FUNCTION_BLOCK FB_Discharger_SFC EXTENDS FB_Object_Template_SFC
VAR_INPUT
	B1: BOOL;
	B2: BOOL;
	dcha_1: BOOL;
	dcha_2: BOOL;
	izda_1: BOOL;
	izda_2: BOOL;
	arriba: BOOL;
	abajo: BOOL;
	cogido: BOOL;
END_VAR
VAR_OUTPUT
	avanza_1: BOOL;
	avanza_2: BOOL;
	baja: BOOL;
	coge: BOOL;
END_VAR
VAR
END_VAR

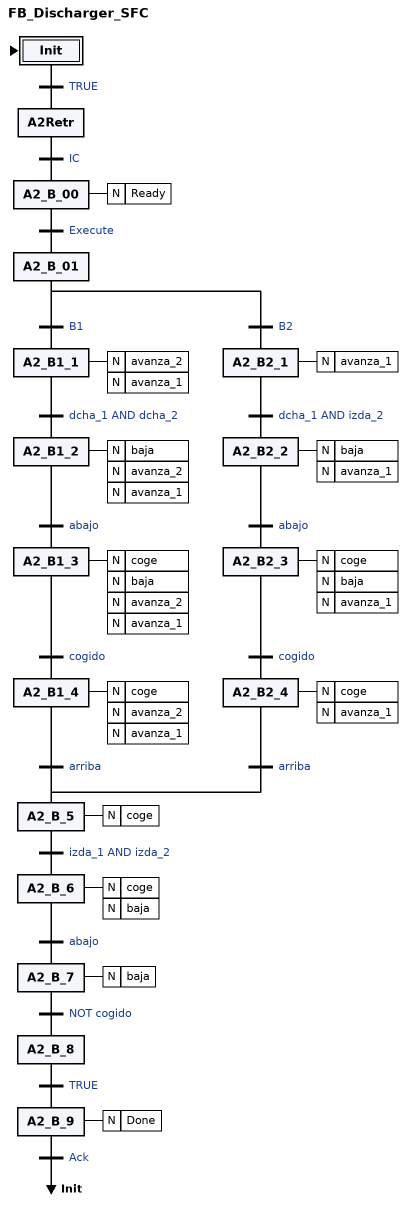
INITIAL_STEP Init:
END_STEP
TRANSITION FROM Init TO A2Retr
    := TRUE;
END_TRANSITION
STEP A2Retr:
END_STEP
TRANSITION FROM A2Retr TO A2_B_00
    := IC;
END_TRANSITION
STEP A2_B_00:
    Ready(N);
END_STEP
TRANSITION FROM A2_B_00 TO A2_B_01
    := Execute;
END_TRANSITION
STEP A2_B_01:
END_STEP
TRANSITION FROM A2_B_01 TO A2_B1_1
    := B1;
END_TRANSITION
STEP A2_B1_1:
    avanza_2(N);
    avanza_1(N);
END_STEP
TRANSITION FROM A2_B1_1 TO A2_B1_2
    := dcha_1 AND dcha_2;
END_TRANSITION
STEP A2_B1_2:
    baja(N);
    avanza_2(N);
    avanza_1(N);
END_STEP
TRANSITION FROM A2_B1_2 TO A2_B1_3
    := abajo;
END_TRANSITION
STEP A2_B1_3:
    coge(N);
    baja(N);
    avanza_2(N);
    avanza_1(N);
END_STEP
TRANSITION FROM A2_B1_3 TO A2_B1_4
    := cogido;
END_TRANSITION
STEP A2_B1_4:
    coge(N);
    avanza_2(N);
    avanza_1(N);
END_STEP
TRANSITION FROM A2_B1_4 TO A2_B_5
    := arriba;
END_TRANSITION
TRANSITION FROM A2_B_01 TO A2_B2_1
    := B2;
END_TRANSITION
STEP A2_B2_1:
    avanza_1(N);
END_STEP
TRANSITION FROM A2_B2_1 TO A2_B2_2
    := dcha_1 AND izda_2;
END_TRANSITION
STEP A2_B2_2:
    baja(N);
    avanza_1(N);
END_STEP
TRANSITION FROM A2_B2_2 TO A2_B2_3
    := abajo;
END_TRANSITION
STEP A2_B2_3:
    coge(N);
    baja(N);
    avanza_1(N);
END_STEP
TRANSITION FROM A2_B2_3 TO A2_B2_4
    := cogido;
END_TRANSITION
STEP A2_B2_4:
    coge(N);
    avanza_1(N);
END_STEP
TRANSITION FROM A2_B2_4 TO A2_B_5
    := arriba;
END_TRANSITION
STEP A2_B_5:
    coge(N);
END_STEP
TRANSITION FROM A2_B_5 TO A2_B_6
    := izda_1 AND izda_2;
END_TRANSITION
STEP A2_B_6:
    coge(N);
    baja(N);
END_STEP
TRANSITION FROM A2_B_6 TO A2_B_7
    := abajo;
END_TRANSITION
STEP A2_B_7:
    baja(N);
END_STEP
TRANSITION FROM A2_B_7 TO A2_B_8
    := NOT cogido;
END_TRANSITION
STEP A2_B_8:
END_STEP
TRANSITION FROM A2_B_8 TO A2_B_9
    := TRUE;
END_TRANSITION
STEP A2_B_9:
    Done(N);
END_STEP
TRANSITION FROM A2_B_9 TO Init
    := Ack;
END_TRANSITION

END_FUNCTION_BLOCK

(* stored: Version 1.1.0.1, ProductVersion 3.1.4024.6
   POU FB_Discharger_SFC: Id {701b0452-272a-4746-924a-7c5e5109a488}, SpecialFunc None *)
